Universal Robots PolyScope program: laengs_greifer_multi_2.urp

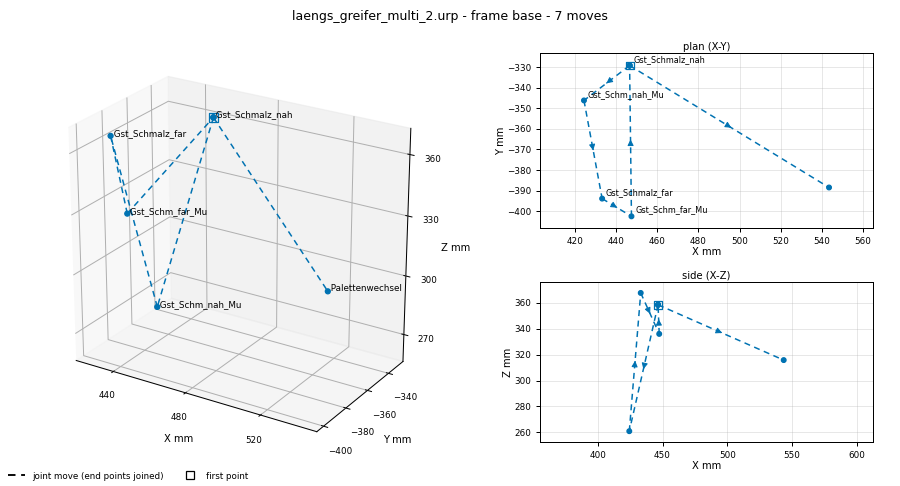
[picture p0: tool path of laengs_greifer_multi_2.urp in frame base, 7 of 42 moves have a stored position in this frame; points joined in program order, loops and branches not executed]
Program laengs_greifer_multi_2 (installation=längs_multi directory=/programs createdIn=5.8.2.10297 lastSavedIn=5.9.5.1031259 robotSerialNumber=20215000780)
Calibrated DH parameters: a=[-0.000076, -0.457222, -0.535711, -0.000049, -0.000015, 0]; d=[0.180847, -379.989416, 320.368416, 59.795924, 0.120055, 0.115601]; alpha=[1.570333, -0.001071, -0.003328, 1.572059, -1.570368, 0]; deltaTheta=[0, 0.727455, -0.372784, -0.354674, 0, 0]
BeforeStart
  Script file /programs/Daten_Bereitstellen.script
    | m_data = rpc_factory("xmlrpc", "http://192.168.0.10:10000")
    | 
    | def DatenAuslesen():
    |   test = m_data.UR_ReadDataFromUsbStick()
    |   return test
    | end
    | 
    | def Dateiname(File):
    |   m_data.UR_SetFileName(File)
    | end
    | 
    | def Palette_Dim():
    |   palette = m_data.UR_Palette()
    |   return palette
    | end
    | 
    | def Karton():
    |   karton = m_data.UR_Karton()
    |   return karton
    | end
    | 
    | def Lagen():
    |   lagen = m_data.UR_Lagen()
    |   return lagen
    | end
    | 
    | def PaketPos(Nummer):
    |   paket_pos = m_data.UR_PaketPos(Nummer)
    |   return paket_pos
    | end
    | 
    | def AnzLagen():
    |   anz_lagen = m_data.UR_AnzLagen()
    |   return anz_lagen
    | end
    | 
    | def AnzPakete():
    |   anz_pakete = m_data.UR_AnzPakete()
    |   return anz_pakete
    | end
    | 
    | def anzPick():
    |   anz_pick = m_data.UR_PaketeZuordnung()
    |   return anz_pick
    | end
    | 
    | def aktStartlage():
    |   lage = m_data.UR_Startlage()
    |   return lage
    | end
    | 
    | def gemKartonhoehe():
    |   hoehe = m_data.UR_Paket_hoehe()
    |   return hoehe
    | end
    | 
    | def liste_ZwischenLagen():
    |   zwLagen = m_data.UR_Zwischenlagen()
    |   return zwLagen
    | end
  SuppressedNode
    Artikel :=  (valueSource=Operator message=Artikelnummer eingeben valueType=String)
  SuppressedNode
    Script: Dateiname(Artikel)
  Artikel_Gewicht := 0.435
  Greifer_Gewicht := 1.7
  Script: set_payload_mass(Greifer_Gewicht)
  Alles_OK := DatenAuslesen()
  Set DigitalOutput pin=licht_start; digitalValue=1
  Set DigitalOutput pin=licht_reset; digitalValue=0
  Set DigitalOutput pin=freigabe_convey; digitalValue=1
  SuppressedNode
    Set DigitalOutput pin=convey_klemmung; digitalValue=1
  SuppressedNode
    URCap SCHMALZ GRIPPER (Schmalz Gripper, J. Schmalz GmbH) dataModel(cmdtype=2)
  Folder Grundeinstellungen
    offset_pickup_z := 40
    SuppressedNode
      URCap SCHMALZ GRIPPER (Schmalz Gripper, J. Schmalz GmbH) dataModel(cmdtype=2)
    URCap Schmalz Gripper (Schmalz Gripper, J.Schmalz GmbH) dataModel(NodeFunctions=2, Variable(key=dummy, variable(name=PartPresentSP2, initializeExpression=False)))
  Folder Variablen Nullen
    liste_paketpos := [0,0,0,0,0,0,0,0,0]
    karton_dim := [0,0,0,0]
    Paket_Zaehler := 0
    signal := False
    Akt_Lifthoehe := 0
    Akt_Lage := 1
    Akt_Lagenart := 1
    Lagenarten := Lagen()
    Zwischenlagen := liste_ZwischenLagen()
    Dicke_ZwLagen := 3
    Akt_Anz_ZwLagen := 0
    Lagenanzahl := AnzLagen()
    Paket_Anzahl := AnzPakete()
    Pick_Anzahl := anzPick()
    Paletten_Masse := Palette_Dim()
    karton_dim := Karton()
    SuppressedNode
      karton_h_gemess :=  (valueSource=Operator message=Bitte gemessene Kartobhöhe in mm eingeben valueType=Integer)
    Script: karton_dim[2]=gemKartonhoehe()
    URCap Schmalz Gripper (Schmalz Gripper, J.Schmalz GmbH)
    kart_hoeh_korre := 0
    offset_basis := 0
    karton_hoehe := karton_dim[2]-kart_hoeh_korre
    einlaufrichtung := karton_dim[3]
    lift_hoehe := Akt_Lifthoehe
    conveyor_start := False
  Folder Startlage
    SuppressedNode
      Paket_Zaehler :=  (valueSource=Operator message=Startpaket Nummer valueType=Integer)
    Akt_Lage := aktStartlage()
Robot Program (runOnlyOnce=false)
  SuppressedNode
    MoveJ speed 60 deg/s, acceleration 80 deg/s^2 (useActiveTCP=true) feature=Palette_extend
      Waypoint Nullpunkt: TCP in base x=289.599 y=-566.564 z=-712.343 mm, rx=-0.0139 ry=-0.0325 rz=-0.7825 rad; joints [312.793, -160.204, -107.825, -90.026, 87.337, 90.018] deg; TCP offset x=-410 y=0 z=-115 mm, rx=0 ry=1.5708 rz=0 rad; feature pose in base x=289.622 y=-566.621 z=-712.344 mm, rx=-0.0027 ry=-0.021 rz=2.3582 rad
      Waypoint Max_auss_re: TCP in base x=-275.386 y=-1063.396 z=-674.131 mm, rx=-0.0139 ry=-0.0325 rz=-0.7826 rad; joints [263.985, -178.789, -37.45, -141.02, 38.649, 88.075] deg
      Waypoint ueber_palett: TCP in base x=-421.858 y=-433.823 z=-216.215 mm, rx=-0.014 ry=-0.0325 rz=-0.7826 rad; joints [241.068, -109.784, -121.165, -122.664, 15.855, 83.941] deg
      Waypoint Max_auss_li: TCP in base x=-1054.914 y=-287.298 z=-669.317 mm, rx=-0.014 ry=-0.0324 rz=-0.7826 rad; joints [203.667, -181.664, -30.299, -152.512, -21.738, 94.073] deg
      Waypoint Max_inn_li: TCP in base x=-560.979 y=208.661 z=-658.157 mm, rx=-0.0139 ry=-0.0325 rz=-0.7826 rad; joints [175.485, -154.81, -111.351, -96.308, -49.976, 91.548] deg
      Waypoint Max_inn_re: TCP in base x=218.479 y=-567.461 z=-662.92 mm, rx=-0.0139 ry=-0.0325 rz=-0.7826 rad; joints [307.399, -155.179, -113.709, -89.156, 81.964, 89.827] deg
  SuppressedNode
    MoveJ speed 60 deg/s, acceleration 80 deg/s^2 (useActiveTCP=true) feature=Base
      Waypoint Null_Aufnahme: TCP in base x=-139.934 y=635.131 z=226.2 mm, rx=-0.0265 ry=-0.0156 rz=-0.8077 rad; joints [116.776, -102.861, -112.441, -146.191, -107.021, 90.331] deg; TCP offset x=-100 y=0 z=-80 mm, rx=0 ry=1.5708 rz=0 rad
  Folder Grundstellung
    MoveJ speed 60 deg/s, acceleration 80 deg/s^2 (useActiveTCP=true positionType=JointAngles) feature=Base
      SuppressedNode
        Waypoint Grund_St: TCP in base x=-489.865 y=390.492 z=244.729 mm, rx=-0.0102 ry=0.003 rz=-0.7688 rad; joints [-55.215, -87.121, 88.987, -1.772, 78.925, 90.279] deg; TCP offset x=-410 y=0 z=-115 mm, rx=0 ry=1.5708 rz=0 rad
      Waypoint Gst_Schmalz_nah: TCP in base x=446.565 y=-329.209 z=358.428 mm, rx=0.0036 ry=0.0001 rz=0.7832 rad; joints [124.272, -84.997, 103.93, 71.181, 90.08, 169.366] deg; TCP offset x=0 y=-51 z=131.4 mm, rx=0 ry=3.1415 rz=0 rad
      SuppressedNode
        Waypoint Gst_Schm_nah_Mu: TCP in base x=423.322 y=-346.599 z=170.08 mm, rx=0.0471 ry=0.0198 rz=2.334 rad; joints [117.61, -72.13, 109.547, 53.577, 92.104, 73.833] deg
      SuppressedNode
        Waypoint Gst_Schmalz_far: TCP in base x=433.21 y=-393.882 z=367.565 mm, rx=0.0111 ry=0.0156 rz=-2.3621 rad; joints [121.386, -94.66, 112.566, -107.207, -89.508, 166.499] deg
      SuppressedNode
        Waypoint Gst_Schm_far_Mu: TCP in base x=501.376 y=-228.647 z=217.522 mm, rx=-0.0928 ry=0.0092 rz=2.3107 rad; joints [130.699, -99.547, 134.849, -129.197, -88.625, 268.032] deg
  conveyor_start := True
  SuppressedNode
    Set DigitalOutput pin=convey_klemmung; digitalValue=1
  Folder Schleife Palette setzen
    Loop While (checkContinuously=false) expression=Akt_Lage<=Lagenanzahl
      Akt_Lagenart := Lagenarten[Akt_Lage-1]
      Folder Start und Endpaket
        If Akt_Lagenart>1
          zaehl_Lageart := 0
          Endpaket := 0
          Loop While (checkContinuously=false) expression=zaehl_Lageart<Akt_Lagenart
            Endpaket := Endpaket+Pick_Anzahl[zaehl_Lageart]
            zaehl_Lageart := zaehl_Lageart+1
          Startpaket := Endpaket-Pick_Anzahl[Akt_Lagenart-1]
        Else 
          Startpaket := 0
          Endpaket := Pick_Anzahl[Akt_Lagenart-1]
        Paket_Zaehler := Startpaket
      Akt_pal_hoehe := (Paletten_Masse[2]/1000)+((karton_hoehe*Akt_Lage)/1000)
      Folder Liftachse fahren
        max_palett_hoeh := 750
        If Akt_pal_hoehe≥(max_palett_hoeh/1000)
          Lagen_ohne_Lift := floor((max_palett_hoeh-Paletten_Masse[2])/karton_hoehe)
          Akt_Lifthoehe := (Akt_Lage-Lagen_ohne_Lift)*(karton_hoehe/1000)
          If Akt_Lifthoehe > 0.900
            Akt_Lifthoehe := 0.900
            SuppressedNode
              Popup Message (haltProgram=false message=Maximale Lifthoehe erreicht inputType=Text)
          Script: move_liftkit(Akt_Lifthoehe*1000)
          lift_hoehe := Akt_Lifthoehe
        Else 
          Script: move_liftkit(0)
      akt_hoe_pick := karton_hoehe-(lift_hoehe*1000)
      Folder Aktuelle Palettenhoehe in Bezug zur Basis
        offset_basis := (0.87+Akt_Lifthoehe)-Akt_pal_hoehe
        If offset_basis>0
          sichere_hoehe := (karton_hoehe/1000)*1.5
        If offset_basis≤0
          sichere_hoehe := (offset_basis*-1)+(karton_hoehe/1000)
      Folder Zwischenlagen zählen
        counter := 0
        Akt_Anz_ZwLagen := 0
        Loop While (checkContinuously=false) expression=counter<Akt_Lage
          Akt_Anz_ZwLagen := Akt_Anz_ZwLagen + Zwischenlagen[counter]
          counter := counter+1
      akt_hoe_ueber := (karton_hoehe*(Akt_Lage-1))-(lift_hoehe*1000)
      akt_hoe_place := (karton_hoehe*Akt_Lage)-(lift_hoehe*1000)+(Akt_Anz_ZwLagen*Dicke_ZwLagen)
      Folder Schleife Lage setzen
        Loop While (checkContinuously=false) expression=Paket_Zaehler<Endpaket
          Folder Paketposition anfragen
            liste_paketpos := PaketPos(Paket_Zaehler)
            If Paket_Zaehler<(Endpaket-1)
              liste_nxt_paket := PaketPos(Paket_Zaehler+1)
              If liste_nxt_paket[4]≤400
                Next_Place_near := True
              Else 
                Next_Place_near := False
            Else 
              Next_Place_near := True
            If einlaufrichtung≟0
              Folder Einlaufrichtung längs
                pickup_x := liste_paketpos[0]
                pickup_y := liste_paketpos[1]
                pickup_z_vor := akt_hoe_pick+offset_pickup_z
                SuppressedNode
                  pickup_z_vor := akt_hoe_pick+kart_hoeh_korre+50
                If liste_paketpos[6]≥2
                  Folder 2 Paket Startposition laengs
                    pickup_rot := d2r(liste_paketpos[2]+90)
                    Vor_Aufn_Pose := p[pickup_x/1000,pickup_y/1000,pickup_z_vor/1000,0,0,pickup_rot]
                    MoveJ speed 120 deg/s, acceleration 160 deg/s^2 (useActiveTCP=true) feature=Aufnahme
                      Waypoint Wegpunkt (Variable): variable=Vor_Aufn_Pose
                    vor_aufn_gelenk := get_actual_joint_positions()
                  Folder 2 Paket laengs aufnehmen
                    Aufn_Pos := p[pickup_x/1000,pickup_y/1000,((akt_hoe_pick-8)/1000),0,0,pickup_rot]
                    Wait DigitalInput pin=digital_in[4]; digitalValue=1
                    URCap Schmalz Gripper (Schmalz Gripper, J.Schmalz GmbH)
                    Wait Sleep waitTime=0.4
                    Wait DigitalInput pin=digital_in[3]; digitalValue=1
                    Wait Sleep waitTime=0.8
                    Wait DigitalInput pin=digital_in[3]; digitalValue=1
                    conveyor_start := False
                    MoveL speed 320 mm/s, acceleration 160 mm/s^2 (useActiveTCP=true) feature=Aufnahme
                      Waypoint Wegpunkt (Variable): variable=Aufn_Pos
                      SuppressedNode
                        Call Greifer_aktivieren_1
                      URCap Schmalz Gripper (Schmalz Gripper, J.Schmalz GmbH)
                    Script: set_payload_mass(Greifer_Gewicht+(Artikel_Gewicht*liste_paketpos[6]))
                    Folder Freifahren Aufnahme
                      tmp_pose_1 := get_actual_tcp_pose()
                      Set DigitalOutput pin=freigabe_convey; digitalValue=0
                      tmp_pose_zwi := pose_trans(tmp_pose_1, p[0,0,0.2,0,0,0])
                      SuppressedNode
                        tmp_pose_zw2 := pose_trans(tmp_pose_1, p[0.02,0.03,0.08,0,0,0])
                      MoveL speed 320 mm/s, acceleration 180 mm/s^2 (useActiveTCP=true) feature=Base
                        Waypoint Wegpunkt (Variable): variable=tmp_pose_zwi
                        SuppressedNode
                          Waypoint Wegpunkt (Variable): variable=tmp_pose_zw2
                      conveyor_start := True
                      Set DigitalOutput pin=freigabe_convey; digitalValue=1
                    Folder Zwischenposition
                      If einlaufrichtung≟1
                        place_rot_ueb := d2r(liste_paketpos[5]-225)
                      Else 
                        place_rot_ueb := d2r(liste_paketpos[5]+45)
                      tmp_pose_1 := get_actual_tcp_pose()
                      pose_zwischen := pose_add(tmp_pose_1, p[-0.360,-0.360,0,0,0,0])
                      Script: pose_zwischen[2]=sichere_hoehe
                      pose_ueb_pal_2 := p[-0.605,-0.570,sichere_hoehe,0,0,place_rot_ueb]
                      SuppressedNode
                        pose_ueb_pal_3 := p[-0.700,-0.108,sichere_hoehe,0,0,place_rot_ueb]
                      SuppressedNode
                        pfosten := p[-0.601,-0.133,sichere_hoehe,0,0,place_rot_ueb]
                      MoveJ speed 180 deg/s, acceleration 180 deg/s^2 (useActiveTCP=true) feature=Base
                        Waypoint Wegpunkt (Variable): variable=pose_zwischen
                        SuppressedNode
                          Waypoint Wegpunkt (Variable): variable=pfosten
                        SuppressedNode
                          Waypoint Wegpunkt (Variable): variable=pose_ueb_pal_3
                        Waypoint Wegpunkt (Variable): variable=pose_ueb_pal_2
                      gelen_ueb_pal_2 := get_actual_joint_positions()
                Else 
                  Folder 1 Paket aufnehmen
                    pickup_rot := d2r(liste_paketpos[2])
                    Vor_Aufn_Pose := p[pickup_x/1000,pickup_y/1000,pickup_z_vor/1000,0,0,pickup_rot]
                    MoveJ speed 180 deg/s, acceleration 120 deg/s^2 (useActiveTCP=true) feature=Aufnahme
                      Waypoint Wegpunkt (Variable): variable=Vor_Aufn_Pose
                    vor_aufn_gelenk := get_actual_joint_positions()
                  Folder 1 Paket quer aufnehmen
                    Aufn_Pos := p[pickup_x/1000,pickup_y/1000,((akt_hoe_pick-8)/1000),0,0,pickup_rot]
                    Wait DigitalInput pin=paket_vorne; digitalValue=1
                    Wait Sleep waitTime=0.1
                    conveyor_start := False
                    MoveL speed 200 mm/s, acceleration 100 mm/s^2 (useActiveTCP=true) feature=Aufnahme
                      Waypoint Wegpunkt (Variable): variable=Aufn_Pos
                      SuppressedNode
                        Call Greifer_aktivieren_1
                      URCap Schmalz Gripper (Schmalz Gripper, J.Schmalz GmbH)
                    Script: set_payload_mass(Greifer_Gewicht+Artikel_Gewicht)
                    Folder Freifahren Aufnahme
                      tmp_pose_1 := get_actual_tcp_pose()
                      tmp_pose_zwi := pose_trans(tmp_pose_1, p[0,0,0.1,0,0,0])
                      SuppressedNode
                        tmp_pose_zw2 := pose_trans(tmp_pose_1, p[0.02,0.03,0.08,0,0,0])
                      MoveL speed 360 mm/s, acceleration 180 mm/s^2 (useActiveTCP=true) feature=Base
                        Waypoint Wegpunkt (Variable): variable=tmp_pose_zwi
                        SuppressedNode
                          Waypoint Wegpunkt (Variable): variable=tmp_pose_zw2
                      conveyor_start := True
                    Folder Zwischenposition
                      If einlaufrichtung≟0
                        place_rot_ueb := d2r(liste_paketpos[5]-225)
                      Else 
                        place_rot_ueb := d2r(liste_paketpos[5]-315)
                      tmp_pose_1 := get_actual_tcp_pose()
                      pose_zwischen := pose_add(tmp_pose_1, p[-0.360,-0.360,sichere_hoehe,0,0,0])
                      Script: pose_zwischen[2]=sichere_hoehe
                      pose_ueb_pal_2 := p[-0.550,-0.650,sichere_hoehe,0,0,place_rot_ueb]
                      SuppressedNode
                        pfosten := p[-0.601,-0.133,sichere_hoehe,0,0,place_rot_ueb]
                      MoveJ speed 180 deg/s, acceleration 120 deg/s^2 (useActiveTCP=true) feature=Base
                        Waypoint Wegpunkt (Variable): motionParameters(blendRadius=0.1); variable=pose_zwischen
                        SuppressedNode
                          Waypoint Wegpunkt (Variable): variable=pfosten
                        Waypoint Wegpunkt (Variable): variable=pose_ueb_pal_2
                      gelen_ueb_pal_2 := get_actual_joint_positions()
            Else 
              Folder Einlaufrichtung quer
                'X und Y vertauscht'
                pickup_x := liste_paketpos[1]*(-1)
                pickup_y := liste_paketpos[0]*(-1)
                pickup_z_vor := akt_hoe_pick+offset_pickup_z
                If liste_paketpos[6]≟1
                  Folder 1 Paket Startposition
                    pickup_rot := d2r(liste_paketpos[2]+90)
                    Vor_Aufn_Pose := p[pickup_x/1000,pickup_y/1000,pickup_z_vor/1000,0,0,pickup_rot]
                    MoveJ speed 180 deg/s, acceleration 160 deg/s^2 (useActiveTCP=true) feature=Aufnahme
                      Waypoint Wegpunkt (Variable): variable=Vor_Aufn_Pose
                    vor_aufn_gelenk := get_actual_joint_positions()
                  Folder 1 Paket aufnehmen
                    Aufn_Pos := p[pickup_x/1000,pickup_y/1000,((akt_hoe_pick)/1000),0,0,pickup_rot]
                    Wait DigitalInput pin=paket_vorne; digitalValue=1
                    Wait Sleep waitTime=0.1
                    SuppressedNode
                      conveyor_start := False
                    MoveL speed 320 mm/s, acceleration 160 mm/s^2 (useActiveTCP=true) feature=Aufnahme
                      Waypoint Wegpunkt (Variable): variable=Aufn_Pos
                      SuppressedNode
                        Call Greifer_aktivieren_1
                      URCap Schmalz Gripper (Schmalz Gripper, J.Schmalz GmbH)
                    Script: set_payload_mass(Greifer_Gewicht+Artikel_Gewicht)
                    Folder Freifahren Aufnahme
                      tmp_pose_1 := get_actual_tcp_pose()
                      tmp_pose_zwi := pose_trans(tmp_pose_1, p[0,0,0.08,0,0,0])
                      MoveL speed 320 mm/s, acceleration 120 mm/s^2 (useActiveTCP=true) feature=Base
                        Waypoint Wegpunkt (Variable): variable=tmp_pose_zwi
                      conveyor_start := True
                    Folder Zwischenposition
                      If einlaufrichtung≟0
                        place_rot_ueb := d2r(liste_paketpos[5]-225)
                      Else 
                        place_rot_ueb := d2r(liste_paketpos[5]-45)
                      tmp_pose_1 := get_actual_tcp_pose()
                      pose_zwischen := pose_add(tmp_pose_1, p[-0.360,-0.360,sichere_hoehe,0,0,0])
                      Script: pose_zwischen[2]=sichere_hoehe
                      pose_ueb_pal_2 := p[-0.600,-0.650,sichere_hoehe,0,0,place_rot_ueb]
                      MoveJ speed 160 deg/s, acceleration 120 deg/s^2 (useActiveTCP=true) feature=Base
                        Waypoint Wegpunkt (Variable): motionParameters(blendRadius=0.1); variable=pose_zwischen
                        Waypoint Wegpunkt (Variable): variable=pose_ueb_pal_2
                      gelen_ueb_pal_2 := get_actual_joint_positions()
                ElseIf liste_paketpos[6]≟2
                  Folder 2 Pakete aufnehmen
                    pickup_rot := d2r(liste_paketpos[2])
                    Vor_Aufn_Pose := p[pickup_x/1000,0,pickup_z_vor/1000,0,0,pickup_rot]
                    MoveJ speed 60 deg/s, acceleration 80 deg/s^2 (useActiveTCP=true) feature=Aufnahme
                      Waypoint Wegpunkt (Variable): variable=Vor_Aufn_Pose
                    vor_aufn_gelenk := get_actual_joint_positions()
                  Folder Erstes Paket aufnehmen
                    Aufn_Pos := p[pickup_x/1000,0,((akt_hoe_pick)/1000),0,0,pickup_rot]
                    Wait DigitalInput pin=paket_vorne; digitalValue=1
                    Wait Sleep waitTime=0.1
                    SuppressedNode
                      conveyor_start := False
                    MoveL speed 320 mm/s, acceleration 120 mm/s^2 (useActiveTCP=true) feature=Aufnahme
                      Waypoint Wegpunkt (Variable): variable=Aufn_Pos
                      SuppressedNode
                        Call Greifer_aktivieren_1
                      URCap Schmalz Gripper (Schmalz Gripper, J.Schmalz GmbH)
                    Script: set_payload_mass(Greifer_Gewicht+Artikel_Gewicht)
                    Folder Zweites Paket aufnehmen
                      Vor_Aufn_Pose := p[pickup_x/1000,((pickup_y/1000)-0.02),pickup_z_vor/1000,0,0,pickup_rot]
                      MoveL speed 320 mm/s, acceleration 120 mm/s^2 (useActiveTCP=true) feature=Aufnahme
                        Waypoint Wegpunkt (Variable): variable=Vor_Aufn_Pose
                      SuppressedNode
                        conveyor_start := True
                      Wait DigitalInput pin=paket_vorne; digitalValue=1
                      URCap Schmalz Gripper (Schmalz Gripper, J.Schmalz GmbH)
                      SuppressedNode
                        Wait Sleep waitTime=0.1
                      SuppressedNode
                        conveyor_start := False
                      Aufn_Pos := p[pickup_x/1000,pickup_y/1000,((akt_hoe_pick)/1000),0,0,pickup_rot]
                      Aufn_Pos_vor := p[pickup_x/1000,pickup_y/1000,pickup_z_vor/1000,0,0,pickup_rot]
                      MoveL speed 320 mm/s, acceleration 120 mm/s^2 (useActiveTCP=true) feature=Aufnahme
                        Waypoint Wegpunkt (Variable): variable=Aufn_Pos_vor
                        Waypoint Wegpunkt (Variable): variable=Aufn_Pos
                      SuppressedNode
                        Call Greifer_deaktivieren_1
                      URCap Schmalz Gripper (Schmalz Gripper, J.Schmalz GmbH) dataModel(NodeFunctions=2, Variable(key=dummy, variable(name=PartPresentSP2, initializeExpression=False)))
                      Wait Sleep waitTime=0.5
                      SuppressedNode
                        Call Greifer_aktivieren_1
                      URCap Schmalz Gripper (Schmalz Gripper, J.Schmalz GmbH)
                      Script: set_payload_mass(Greifer_Gewicht+(Artikel_Gewicht*2))
                    Folder Freifahren
                      tmp_pose_1 := get_actual_tcp_pose()
                      tmp_pose_zwi := pose_trans(tmp_pose_1, p[0,0,0.08,0,0,0])
                      MoveL speed 160 mm/s, acceleration 60 mm/s^2 (useActiveTCP=true) feature=Base
                        Waypoint Wegpunkt (Variable): variable=tmp_pose_zwi
                      conveyor_start := True
                    Folder Zwischenposition
                      place_rot_ueb := d2r(liste_paketpos[5]+135)
                      tmp_pose_1 := get_actual_tcp_pose()
                      pose_zwischen := pose_add(tmp_pose_1, p[-0.360,-0.360,0,0,0,0])
                      Script: pose_zwischen[2]=sichere_hoehe
                      pose_ueb_pal_2 := p[-0.600,-0.650,sichere_hoehe,0,0,place_rot_ueb]
                      MoveJ speed 90 deg/s, acceleration 60 deg/s^2 (useActiveTCP=true) feature=Base
                        Waypoint Wegpunkt (Variable): variable=pose_zwischen
                        Waypoint Wegpunkt (Variable): variable=pose_ueb_pal_2
                      gelen_ueb_pal_2 := get_actual_joint_positions()
                ElseIf liste_paketpos[6]≟3
                  Folder 3 Pakete aufnehmen
                    pickup_rot := d2r(liste_paketpos[2])
                    Vor_Aufn_Pose := p[pickup_x/1000,karton_dim[1]/2000,pickup_z_vor/1000,0,0,pickup_rot]
                    MoveJ speed 60 deg/s, acceleration 80 deg/s^2 (useActiveTCP=true) feature=Aufnahme
                      Waypoint Wegpunkt (Variable): variable=Vor_Aufn_Pose
                    vor_aufn_gelenk := get_actual_joint_positions()
                  Folder Erstes Paket aufnehmen
                    Aufn_Pos := p[pickup_x/1000,karton_dim[1]/2000,((akt_hoe_pick)/1000),0,0,pickup_rot]
                    Wait DigitalInput pin=paket_vorne; digitalValue=1
                    Wait Sleep waitTime=0.1
                    MoveL speed 160 mm/s, acceleration 80 mm/s^2 (useActiveTCP=true) feature=Aufnahme
                      Waypoint Wegpunkt (Variable): variable=Aufn_Pos
                      SuppressedNode
                        Call Greifer_aktivieren_1
                      URCap Schmalz Gripper (Schmalz Gripper, J.Schmalz GmbH)
                    Script: set_payload_mass(Greifer_Gewicht+Artikel_Gewicht)
                    Folder Zweites Paket aufnehmen
                      Vor_Aufn_Pose := p[pickup_x/1000,(-1*((karton_dim[1]/2000)+0.01)),pickup_z_vor/1000,0,0,pickup_rot]
                      MoveL speed 160 mm/s, acceleration 80 mm/s^2 (useActiveTCP=true) feature=Aufnahme
                        Waypoint Wegpunkt (Variable): variable=Vor_Aufn_Pose
                      Wait DigitalInput pin=paket_vorne; digitalValue=1
                      Aufn_Pos := p[pickup_x/1000,(-1*(karton_dim[1]/2000)),((akt_hoe_pick)/1000),0,0,pickup_rot]
                      Vor_Aufn_Pose := p[pickup_x/1000,(-1*(karton_dim[1]/2000)),pickup_z_vor/1000,0,0,pickup_rot]
                      MoveL speed 160 mm/s, acceleration 80 mm/s^2 (useActiveTCP=true) feature=Aufnahme
                        Waypoint Wegpunkt (Variable): variable=Vor_Aufn_Pose
                        Waypoint Wegpunkt (Variable): variable=Aufn_Pos
                      SuppressedNode
                        Call Greifer_deaktivieren_1
                      URCap Schmalz Gripper (Schmalz Gripper, J.Schmalz GmbH) dataModel(NodeFunctions=2)
                      Wait Sleep waitTime=0.1
                      SuppressedNode
                        Call Greifer_aktivieren_1
                      URCap Schmalz Gripper (Schmalz Gripper, J.Schmalz GmbH)
                      Script: set_payload_mass(Greifer_Gewicht+(Artikel_Gewicht*2))
                    Folder Drittes Paket aufnehmen
                      Vor_Aufn_Pose := p[pickup_x/1000,(-1*((karton_dim[1]*1.5/1000)+0.01)),pickup_z_vor/1000,0,0,pickup_rot]
                      MoveL speed 160 mm/s, acceleration 80 mm/s^2 (useActiveTCP=true) feature=Aufnahme
                        Waypoint Wegpunkt (Variable): variable=Vor_Aufn_Pose
                      Wait DigitalInput pin=paket_vorne; digitalValue=1
                      Aufn_Pos := p[pickup_x/1000,(-1*(karton_dim[1]*1.5/1000)),((akt_hoe_pick)/1000),0,0,pickup_rot]
                      MoveL speed 160 mm/s, acceleration 80 mm/s^2 (useActiveTCP=true) feature=Aufnahme
                        Waypoint Wegpunkt (Variable): variable=Aufn_Pos
                      SuppressedNode
                        Call Greifer_deaktivieren_1
                      URCap Schmalz Gripper (Schmalz Gripper, J.Schmalz GmbH) dataModel(NodeFunctions=2)
                      Wait Sleep waitTime=0.1
                      SuppressedNode
                        Call Greifer_aktivieren_1
                      URCap Schmalz Gripper (Schmalz Gripper, J.Schmalz GmbH)
                      Script: set_payload_mass(Greifer_Gewicht+(Artikel_Gewicht*3))
                    Folder Freifahren
                      tmp_pose_1 := get_actual_tcp_pose()
                      tmp_pose_zwi := pose_trans(tmp_pose_1, p[0,0,0.08,0,0,0])
                      MoveL speed 160 mm/s, acceleration 60 mm/s^2 (useActiveTCP=true) feature=Base
                        Waypoint Wegpunkt (Variable): variable=tmp_pose_zwi
                      conveyor_start := True
                    Folder Zwischenposition
                      place_rot_ueb := d2r(liste_paketpos[5]+135)
                      tmp_pose_1 := get_actual_tcp_pose()
                      pose_zwischen := pose_add(tmp_pose_1, p[-0.360,-0.360,sichere_hoehe,0,0,0])
                      pose_ueb_pal_2 := p[-0.600,-0.650,sichere_hoehe,0,0,place_rot_ueb]
                      MoveJ speed 90 deg/s, acceleration 60 deg/s^2 (useActiveTCP=true) feature=Base
                        Waypoint Wegpunkt (Variable): motionParameters(blendRadius=0.1); variable=pose_zwischen
                        Waypoint Wegpunkt (Variable): variable=pose_ueb_pal_2
                      gelen_ueb_pal_2 := get_actual_joint_positions()
          Folder Paket ablegen
            place_x := liste_paketpos[3]*(-1)
            place_y := liste_paketpos[4]*(-1)
            place_z := akt_hoe_place
            If Akt_Lage≤6
              place_z := akt_hoe_place+3
            If einlaufrichtung≟1
              SuppressedNode
                place_rot := d2r(liste_paketpos[5]-90)
              If liste_paketpos[6]≟1
                place_rot := d2r(liste_paketpos[5])
              Else 
                place_rot := d2r(liste_paketpos[5]-90)
            Else 
              If liste_paketpos[6]≟1
                place_rot := d2r(liste_paketpos[5])
              Else 
                place_rot := d2r(liste_paketpos[5]+90)
            place_pos := p[place_x/1000,place_y/1000,(place_z/1000),0,0,place_rot]
            x_vec := liste_paketpos[7]
            y_vec := liste_paketpos[8]
            place_x_vor := place_x+(x_vec*50*(-1))
            place_y_vor := place_y+(y_vec*50*(-1))
            place_z_vor := place_z+karton_hoehe+30
            place_pos_vor := p[place_x_vor/1000,place_y_vor/1000,place_z_vor/1000,0,0,place_rot]
            Folder Debug Drehwinkel
              rot_debug_2 := pose_trans(Palette_extend, place_pos_vor)
              rot_debug_trans := get_inverse_kin(rot_debug_2)
              If rot_debug_trans[5]≥6
                Script: rot_debug_trans[5]=rot_debug_trans[5]-6.28318
              If rot_debug_trans[5]≤-6
                Script: rot_debug_trans[5]=rot_debug_trans[5]+6.28318
            SuppressedNode
              Popup Message (haltProgram=false inputType=Variable) variable=rot_debug_trans
            SuppressedNode
              MoveJ speed 60 deg/s, acceleration 80 deg/s^2 (useActiveTCP=true) feature=Palette_extend
                Waypoint Wegpunkt (Variable): variable=place_pos_vor
            Script: movej(rot_debug_trans, a=2, v=3.14)
            MoveL speed 120 mm/s, acceleration 800 mm/s^2 (useActiveTCP=true) feature=Palette_extend
              Waypoint Wegpunkt (Variable): variable=place_pos
            SuppressedNode
              Call Greifer_deaktivieren_1
            URCap Schmalz Gripper (Schmalz Gripper, J.Schmalz GmbH) dataModel(NodeFunctions=2)
            Script: set_payload_mass(Greifer_Gewicht)
            Folder Freifahren Ablage
              tmp_pose_1 := get_actual_tcp_pose()
              tmp_pose_ablage := pose_trans(tmp_pose_1, p[0,0,0.030,0,0,0])
              MoveL speed 60 mm/s, acceleration 80 mm/s^2 (useActiveTCP=true) feature=Base
                Waypoint Wegpunkt (Variable): variable=tmp_pose_ablage
            Folder Zurueck zur Aufnahmeposition
              Script: movej(gelen_ueb_pal_2, a=2, v=3.141)
              If Next_Place_near≟ True
                If liste_nxt_paket[6]≟1
                  MoveJ speed 180 deg/s, acceleration 120 deg/s^2 (useActiveTCP=true positionType=JointAngles) feature=Base
                    Waypoint Gst_Schmalz_nah: TCP in base x=446.565 y=-329.209 z=358.428 mm, rx=0.0036 ry=0.0001 rz=0.7832 rad; joints [124.272, -84.997, 103.93, 71.181, 90.08, 169.366] deg
                    SuppressedNode
                      Waypoint Gst_Schm_nah_Mu: TCP in base x=-442.893 y=485.402 z=203.694 mm, rx=0 ry=0 rz=-2.3819 rad; joints [-64.489, -69.302, 101.415, 57.859, 90.268, 161.908] deg
                Else 
                  MoveJ speed 180 deg/s, acceleration 120 deg/s^2 (useActiveTCP=true positionType=JointAngles) feature=Base
                    Waypoint Gst_Schm_nah_Mu: TCP in base x=424.385 y=-346.169 z=260.946 mm, rx=0.0445 ry=0.0186 rz=2.3338 rad; joints [117.622, -76.916, 105.194, 62.717, 92.125, 73.867] deg
                    SuppressedNode
                      Waypoint Gst_Schmalz_nah: TCP in base x=-324.647 y=485.387 z=236.052 mm, rx=-0.0048 ry=0.0011 rz=2.3577 rad; joints [-68.857, -73.375, 103.379, 60.159, 90.385, -114.011] deg
              Else 
                If liste_nxt_paket[6]≟1
                  MoveJ speed 180 deg/s, acceleration 120 deg/s^2 (useActiveTCP=true positionType=JointAngles) feature=Base
                    Waypoint Gst_Schmalz_far: TCP in base x=433.21 y=-393.882 z=367.565 mm, rx=0.0111 ry=0.0156 rz=-2.3621 rad; joints [121.386, -94.66, 112.566, -107.207, -89.508, 166.499] deg
                    SuppressedNode
                      Waypoint Gst_Schm_far_Mu: TCP in base x=501.376 y=-228.647 z=217.522 mm, rx=-0.0928 ry=0.0092 rz=2.3107 rad; joints [130.699, -99.547, 134.849, -129.197, -88.625, 268.032] deg
                Else 
                  MoveJ speed 180 deg/s, acceleration 120 deg/s^2 (useActiveTCP=true positionType=JointAngles) feature=Base
                    Waypoint Gst_Schm_far_Mu: TCP in base x=447.464 y=-402.502 z=335.972 mm, rx=-0.0736 ry=0.0258 rz=2.3189 rad; joints [115.69, -98.774, 120.462, -114.955, -88.905, 252.649] deg
                    SuppressedNode
                      Waypoint Gst_Schmalz_far: TCP in base x=433.21 y=-393.882 z=367.565 mm, rx=0.0111 ry=0.0156 rz=-2.3621 rad; joints [121.386, -94.66, 112.566, -107.207, -89.508, 166.499] deg
          Paket_Zaehler := Paket_Zaehler+1
      If Zwischenlagen[Akt_Lage-1]≟1
        signal := True
        Popup Message (haltProgram=false message=Zwischenlage einlegen und dann WEITER drücken! Achtung Roboter fährt los! inputType=Text)
        signal := False
      MoveJ speed 60 deg/s, acceleration 80 deg/s^2 (useActiveTCP=true positionType=JointAngles) feature=Base
        Waypoint Gst_Schmalz_nah: TCP in base x=446.565 y=-329.209 z=358.428 mm, rx=0.0036 ry=0.0001 rz=0.7832 rad; joints [124.272, -84.997, 103.93, 71.181, 90.08, 169.366] deg
      Akt_Lage := Akt_Lage+1
    MoveJ speed 60 deg/s, acceleration 80 deg/s^2 (useActiveTCP=true) feature=Base
      Waypoint Palettenwechsel: TCP in base x=543.47 y=-388.474 z=315.779 mm, rx=0.0048 ry=0.0149 rz=0.8721 rad; joints [128.733, -72.84, 93.685, 69.526, 90.853, 168.738] deg
    URCap LIFTKIT (LIFTKIT, SKF Actuation System (Liestal) AG) dataModel(position=0)
    signal := True
    Popup Message (haltProgram=false message=Palette wechseln und dann WEITER drücken! Achtung Roboter fährt los! inputType=Text)
    signal := False
    Akt_Lage := 1
    lift_hoehe := 0
    Akt_Lifthoehe := 0
Thread Thread_1 (runOnlyOnce=false)
  If einlaufrichtung≟1
    If conveyor_start≟ True
      Set DigitalOutput pin=freigabe_convey; digitalValue=1
      Set DigitalOutput pin=klemmung; digitalValue=1
      If paket_vorne≟  False
        Set DigitalOutput pin=klemmung; digitalValue=0
        Wait DigitalInput pin=digital_in[3]; digitalValue=1
        Set DigitalOutput pin=klemmung; digitalValue=1
        Wait DigitalInput pin=digital_in[4]; digitalValue=1
    Else 
      Set DigitalOutput pin=freigabe_convey; digitalValue=0
  Script: sync()
Thread Thread_2 (runOnlyOnce=false)
  'Signalleuchte Zwischenlage'
  If signal≟ True
    Set DigitalOutput pin=licht_stopp; digitalValue=1
    Set DigitalOutput pin=licht_start; digitalValue=1
    Set DigitalOutput pin=digital_out[6]; digitalValue=1
    Wait Sleep waitTime=0.2
    Set DigitalOutput pin=licht_stopp; digitalValue=0
    Set DigitalOutput pin=licht_start; digitalValue=0
    Set DigitalOutput pin=digital_out[6]; digitalValue=0
    Wait Sleep waitTime=0.2
  Else 
    Set DigitalOutput pin=licht_stopp; digitalValue=0
    Set DigitalOutput pin=licht_start; digitalValue=0
    Set DigitalOutput pin=digital_out[6]; digitalValue=0
  Script: sync()
SuppressedNode
  SubProgram -> Greifer_deaktivieren_1
SuppressedNode
  SubProgram -> Greifer_aktivieren_1
SubProgram Greifer_aktivieren_1 (keepSynchronizedWithDisk=false) programFile=/programs/Greifer_aktivieren.urp
  URCap SCHMALZ GRIPPER (Schmalz Gripper, J. Schmalz GmbH) dataModel(cmdtype=0, wait_h2=1)
SubProgram Greifer_deaktivieren_1 (keepSynchronizedWithDisk=false) programFile=/programs/Greifer_deaktivieren.urp
  URCap SCHMALZ GRIPPER (Schmalz Gripper, J. Schmalz GmbH) dataModel(wait_h2=0, cmdtype=2)
  URCap SCHMALZ GRIPPER (Schmalz Gripper, J. Schmalz GmbH) dataModel(releasetime=200, wait_h2=0, cmdtype=1)
  URCap SCHMALZ GRIPPER (Schmalz Gripper, J. Schmalz GmbH) dataModel(wait_h2=0, cmdtype=2)
